// TIA Portal V16 export
// export: Created 2024-12-03T15:41:43.4350432Z, ExportSetting WithDefaults, DisplayName Totally Integrated Automation Portal, DisplayVersion V16 Update 6, DisplayName TIA Portal Version Control Interface, DisplayVersion V16 Update 2, DisplayName TIA Portal Openness, DisplayVersion V16 Update 6, DisplayName TIA Portal Teamcenter Gateway, DisplayVersion V16, DisplayName SINAMICS Startdrive Advanced, DisplayVersion V16 Update 5, DisplayName SINAMICS Startdrive G130, G150, S120, S150, SINAMICS MV, S210, DisplayVersion V16 Update 5, DisplayName SINAMICS Startdrive G110M, G120, G120C, G120D, G120P, G115D, DisplayVersion V16 Update 5, DisplayName STEP 7 Professional, DisplayVersion V16 Update 6, DisplayName STEP 7 Safety, DisplayVersion V16, DisplayName WinCC Advanced / Unified PC, DisplayVersion V16 Update 6
FUNCTION_BLOCK "TrafficController_INTERSECT_RECEIVE_PRIO_FB"   // FB86, SCL
{ S7_Optimized_Access := 'TRUE' }
VERSION : 0.1
// intersection receives from one section and can sent to other 3 sections
// stored: AutoNumber true, IsIECCheckEnabled false, IsRetainMemResEnabled false, MemoryReserve 100, SetENOAutomatically false, UDAEnableTagReadback false
   VAR_INPUT
      I_SendingConveyor_1 { ExternalAccessible := 'False'; ExternalVisible := 'False'; ExternalWritable := 'False'} : "Conveyor_UDT";   // The main conveyor on the intersection
      I_SendingConveyor_2 : "Conveyor_UDT";
      I_IntersectionConveyor : "Conveyor_UDT";
      I_Option_1_Settings { ExternalAccessible := 'False'; ExternalVisible := 'False'; ExternalWritable := 'False'} : "Intersection";   // Intersection settings for option 1 (no split executed)
      I_Option_2_Settings { ExternalAccessible := 'False'; ExternalVisible := 'False'; ExternalWritable := 'False'} : "Intersection";   // Intersection settings for option 2 (split executed)
   END_VAR
   VAR_OUTPUT
      O_AccumulateConv_1 : Bool;
      O_AccumulateConv_2 : Bool;
   END_VAR
   VAR_IN_OUT
      IO_IntersectionSettings : "Intersection";
   END_VAR
   VAR
      option : Int;
      OptionsSaved : Bool;
   END_VAR
BEGIN
   #O_AccumulateConv_1 := TRUE;
   #O_AccumulateConv_2 := TRUE;

   REGION FLOW CONTROL

       #option := 0;

       IF #I_SendingConveyor_1.Status.RequestForSending AND #I_IntersectionConveyor.Status.Empty THEN
           #option := 1;
       END_IF;

       IF NOT #I_SendingConveyor_1.Status.RequestForSending AND
           #I_SendingConveyor_2.Status.RequestForSending AND
           #I_IntersectionConveyor.Status.Empty THEN
           #option := 2;
       END_IF;

   END_REGION

   REGION CHECK TO TRANSFER SETTINGS

       IF (#I_SendingConveyor_1.Status.RequestForSending OR #I_SendingConveyor_2.Status.RequestForSending)
           AND #I_IntersectionConveyor.Status.Empty THEN

           CASE #option OF
               1:
                   #IO_IntersectionSettings := #I_Option_1_Settings;
               2:
                   #IO_IntersectionSettings := #I_Option_2_Settings;
           END_CASE;


       END_IF;

   END_REGION

   REGION TURN OFF ACCUMULATION OF SENDING CONV

       IF (#I_SendingConveyor_1.Status.RequestForSending OR #I_SendingConveyor_2.Status.RequestForSending)
           AND #I_IntersectionConveyor.Status.Empty THEN

           IF #option = 1 THEN
               #O_AccumulateConv_1 := FALSE;
           END_IF;

           IF #option = 2 THEN
               #O_AccumulateConv_2 := FALSE;
           END_IF;

       END_IF;

   END_REGION
END_FUNCTION_BLOCK
